Staubli VAL3: onStart.pgx

program onStart()
  local num i
  local string l_sMessage
begin
  // logMsg
  logMsg("[KERNEL] INTERFACE:PAGE TOOL")
  // be aware these value will change all the value
  call language:message(l_sMessage,129)
  popUpMsg(l_sMessage)
  // set the tool as default
  nIndexTool=saveData:nIndexTool
  // reset the Key pressure
  call use:nullKey(nKey)
  // define the list
  call buildList()
  // build the page
  call refreshStatic()
  // define the list
end
